FUNCTION_BLOCK FB_Observable_UINT EXTENDS FB_AbstractObservable
VAR
    _nVal:              UINT;
END_VAR

METHOD  Notify : I_Observable
VAR
    i:      UDINT;
END_VAR
Notify := THIS^;

IF THIS^.nObserverCount <= 0 THEN
    RETURN;
END_IF

FOR i := 0 TO THIS^.nLastIdx DO
    THIS^.pipObserver[i].Update(THIS^._nVal);
END_FOR
END_METHOD

METHOD  NotifyLast : I_Observable
NotifyLast := THIS^;

IF THIS^.nObserverCount <= 0 THEN
    RETURN;
END_IF

THIS^.pipObserver[THIS^.nLastIdx].Update(THIS^._nVal);
END_METHOD

PROPERTY nValue16 : UINT
GET
nValue16 := THIS^._nVal;
END_GET
SET
THIS^._nVal := nValue16;

IF THIS^._bAutoNotify THEN
    THIS^.Notify();
END_IF
END_SET
END_PROPERTY

END_FUNCTION_BLOCK

(* stored: Version 1.1.0.1, ProductVersion 3.1.4024.12
   POU FB_Observable_UINT: Id {f2d7fe92-4d1e-47f3-bc2f-43e40068362f}, SpecialFunc None
   Method Notify: Id {e877583d-d78e-4b21-a98f-6f809b093685}
   Method NotifyLast: Id {d479e08c-8f99-42ea-a71a-fe3a3806deb4}
   Property nValue16: Id {af502dac-a26d-48ef-8a2d-4ee091e8d385}
   Get Get: Id {f747421d-9861-4e67-82a8-164d0b8556a2}
   Set Set: Id {1715d78f-c08f-4f38-91ae-928e9c0a47c7} *)
